// TIA Portal V17 export
// export: Created 2022-07-28T18:03:03.6741097Z, ExportSetting None, DisplayName Totally Integrated Automation Portal, DisplayVersion V17, DisplayName TIA Portal Openness, DisplayVersion V17, DisplayName TIA Portal Teamcenter Gateway, DisplayVersion V17, DisplayName TIA Portal Version Control Interface, DisplayVersion V17, DisplayName TIA Portal Test Suite Advanced, DisplayVersion V17, DisplayName SINAMICS Startdrive Advanced, DisplayVersion V17, DisplayName SINAMICS DCC, DisplayVersion V17, DisplayName SINAMICS Startdrive G130, G150, S120, S150, SINAMICS MV, S210, DisplayVersion V17, DisplayName SINAMICS Startdrive G110M, G120, G120C, G120D, G120P, G115D, DisplayVersion V17, DisplayName STEP 7 Professional, DisplayVersion V17, DisplayName SIMATIC Energy Suite, DisplayVersion V17, DisplayName STEP 7 CFC, DisplayVersion V17, DisplayName STEP 7 Safety, DisplayVersion V17, DisplayName WinCC Advanced / Unified PC, DisplayVersion V17, DisplayName SIMATIC Visualization Architect, DisplayVersion V17
DATA_BLOCK "D_General_HMI"   // DB12
TITLE = GenHMI
{ S7_Optimized_Access := 'TRUE' }
// General data for exchange with HMI (AW, CMD, SP, ect.)
// stored: MemoryReserve 100
   VAR
      i_CMD : Int;   // Gener command
      w_MW1 { ExternalWritable := 'False'} : Word;   // Message word 1
      w_MW2 { ExternalWritable := 'False'} : Word := 16#0;   // Message word 2
      w_MW3 { ExternalWritable := 'False'} : Word := 16#0;   // Message word 3
      w_MW4 { ExternalWritable := 'False'} : Word := 16#0;   // Message word 4
      w_MW5 { ExternalWritable := 'False'} : Word := 16#0;   // Message word 5
      w_MW6 { ExternalWritable := 'False'} : Word := 16#0;   // Message word 6
      w_MW7 { ExternalWritable := 'False'} : Word := 16#0;   // Message word 7
      w_MW8 { ExternalWritable := 'False'} : Word := 16#0;   // Message word 8
      w_MW9 { ExternalWritable := 'False'} : Word := 16#0;   // Message word 9
      w_MW10 { ExternalWritable := 'False'} : Word := 16#0;   // Message word 10
   END_VAR
BEGIN
END_DATA_BLOCK
